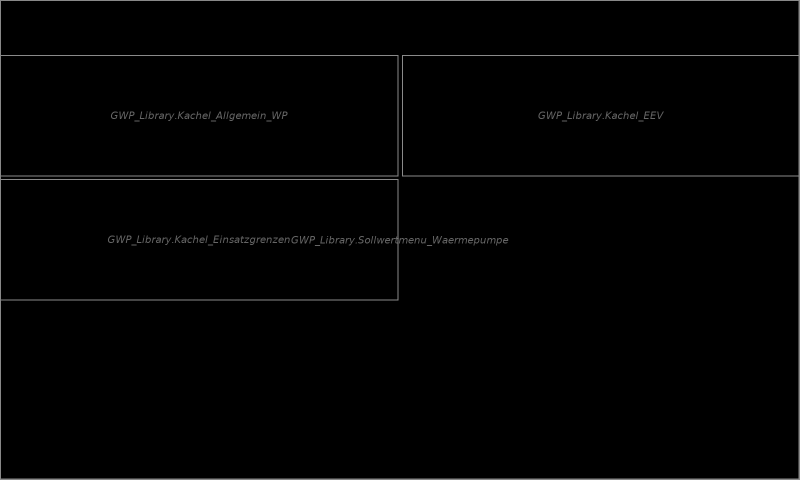
VISUALIZATION Sollwertmenu_Waermepumpe  // 800x480
    Frame (0,0 800x480)
        shows GWP_Library.Sollwertmenu_Waermepumpe(FB_Init_1 := Main.Init_0)
    Frame (402,55 398x121)
        shows GWP_Library.Kachel_EEV()
        OnMouseClick: change screen: EEv
    Frame (0,179 398x121)
        shows GWP_Library.Kachel_Einsatzgrenzen()
        OnMouseClick: change screen: EG_Innen
    Frame (0,55 398x121)
        shows GWP_Library.Kachel_Allgemein_WP()
        OnMouseClick: change screen: Kreis_3KO_SollwerteAllg
END_VISUALIZATION

(* stored: Version 1.1.0.1, ProductVersion 3.1.4022.6
   Visu Sollwertmenu_Waermepumpe: Id {8cba2575-7eeb-466b-bd59-a42389688c4b} *)
